INTERFACE I_Axis

METHOD EndOfCycle : BOOL
VAR_INPUT
END_VAR
END_METHOD

METHOD Run : BOOL
VAR_INPUT
END_VAR
END_METHOD

PROPERTY stAxis : REFERENCE TO ST_AxisStruct
GET
END_GET
SET
END_SET
END_PROPERTY

END_INTERFACE

(* stored: Version 1.1.0.1, ProductVersion 3.1.4024.12
   Itf I_Axis: Id {aa3f26f1-e1dd-43e1-ad72-924a566d91d1}
   Method EndOfCycle: Id {1e7d03ee-b03d-4e24-bc82-27dce521a52e}
   Method Run: Id {7e3148d5-8f02-43cd-bfcb-03545931b5e8}
   Property stAxis: Id {c7710a62-b9e1-478e-bbd1-1fb2fb0a2fc5}
   Get Get: Id {86849ae3-b1b2-4c86-b3ef-f5c9ef8278d9}
   Set Set: Id {cddb2d57-7d29-4e35-beef-82c9ff08c26e} *)
